PROGRAM TICK
VAR
	ins : BOOL;
	et : TIME;
	tick: TON;
	canGrabTableData: BOOL := FALSE;
	
	nDayOfTheWeek : INT := 1;
	
	tdSimTime : TOD := TOD#4:0:0;
	SimTime : UDINT;
	
	// Traffic flow time index for CONSTANTS.aTrafficFlowTimes
	x1i : INT := 1;
	x2i : INT := 2;
	x1 : REAL := TOD_TO_REAL(CONSTANTS.aTrafficFlowTimes[x1i]);
	x2 : REAL := TOD_TO_REAL(CONSTANTS.aTrafficFlowTimes[x2i]);

	tdTickTime : TOD := TOD#0:15:0;
END_VAR
VAR // added by the converter: edge detectors and wires of the graphical bodies
    _w1, _w2, _w3 : BOOL;
END_VAR

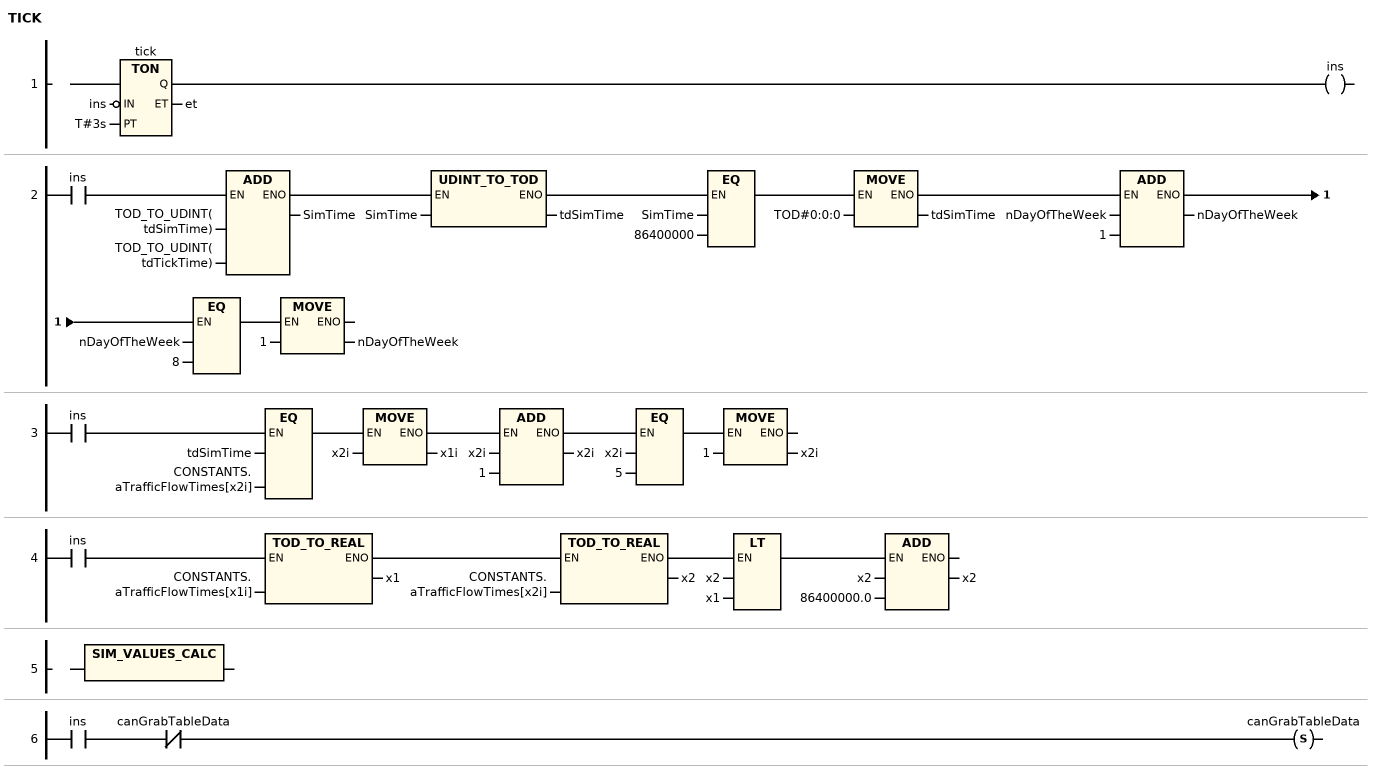
// NETWORK 1
tick(IN := NOT ins, PT := T#3s, ET => et); // TON
ins := tick.Q;

// NETWORK 2
_w1 := ins;
IF _w1 THEN SimTime := (TOD_TO_UDINT(tdSimTime)) + (TOD_TO_UDINT(tdTickTime)); END_IF
IF _w1 THEN tdSimTime := UDINT_TO_TOD(SimTime); END_IF
IF _w1 AND SimTime = 86400000 THEN tdSimTime := TOD#0:0:0; END_IF
IF _w1 AND SimTime = 86400000 THEN nDayOfTheWeek := nDayOfTheWeek + 1; END_IF
IF _w1 AND SimTime = 86400000 AND nDayOfTheWeek = 8 THEN nDayOfTheWeek := 1; END_IF

// NETWORK 3
_w2 := ins AND tdSimTime = CONSTANTS.aTrafficFlowTimes[x2i];
IF _w2 THEN x1i := x2i; END_IF
IF _w2 THEN x2i := x2i + 1; END_IF
IF _w2 AND x2i = 5 THEN x2i := 1; END_IF

// NETWORK 4
_w3 := ins;
IF _w3 THEN x1 := TOD_TO_REAL(CONSTANTS.aTrafficFlowTimes[x1i]); END_IF
IF _w3 THEN x2 := TOD_TO_REAL(CONSTANTS.aTrafficFlowTimes[x2i]); END_IF
IF _w3 AND x2 < x1 THEN x2 := x2 + 86400000.0; END_IF

// NETWORK 5
SIM_VALUES_CALC();

// NETWORK 6
canGrabTableData S= ins AND NOT canGrabTableData;

END_PROGRAM

(* stored: Version 1.1.0.1, ProductVersion 3.1.4024.12
   POU TICK: Id {37d78b7f-dc72-4185-adb8-49490fffb64d}, SpecialFunc None *)
